FUNCTION_BLOCK MotorControla
VAR_INPUT
	Premik: BOOL;
	Smer: BOOL;
	Select: BOOL;
	KS: BOOL;
	Step: BOOL;
	Limes: WORD;
END_VAR
VAR_OUTPUT
	OutPremik: BOOL;
	OutSmer: BOOL;
	Interlock: BOOL;
	Stop: BOOL;
	Position: WORD;
END_VAR
VAR
	R_TRIG_0: R_TRIG;
	Dump: TIME;
	InL: TOF;
	RS_0: RS;

	R_TRIG_1: R_TRIG;
	TON0: TON;
	TON1: TON;
	TON_0: TON;
	Counter_0: Counter;
	F_TRIG_0: F_TRIG;
	InL1: TOF;
	IntL1: BOOL;
	IntL2: BOOL;
	IntL3: BOOL;
	R_TRIG_2: R_TRIG;
END_VAR
//dODAJ COLLISION DETECTION AND AVOIDANCE
//ZRIHTAJ SMER, KI SE SLABO SPREMINJA

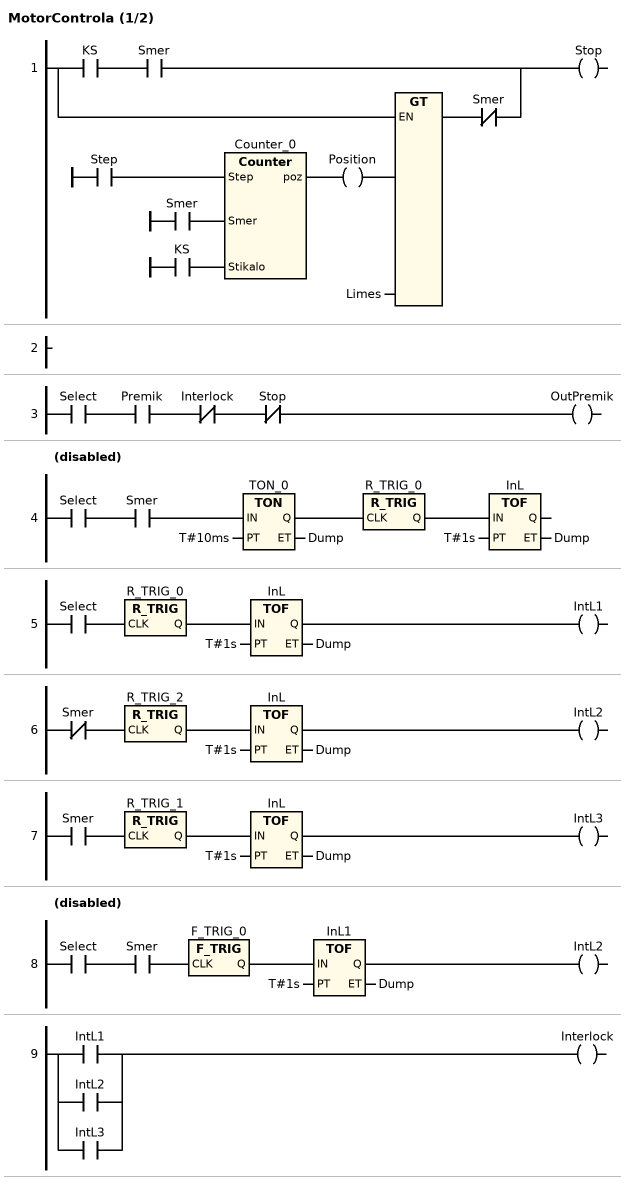
// NETWORK 1
Counter_0(Step := Step, Smer := Smer, Stikalo := KS); // Counter
Position := Counter_0.poz;
Stop := KS AND Smer OR Counter_0.poz > Limes AND NOT Smer;

// NETWORK 2

// NETWORK 3
OutPremik := Select AND Premik AND NOT Interlock AND NOT Stop;

// NETWORK 4 (disabled)
// TON_0(IN := Select AND Smer, PT := T#10ms, ET => Dump); // TON
// R_TRIG_0(CLK := TON_0.Q); // R_TRIG
// InL(IN := R_TRIG_0.Q, PT := T#1s, ET => Dump); // TOF

// NETWORK 5
R_TRIG_0(CLK := Select); // R_TRIG
InL(IN := R_TRIG_0.Q, PT := T#1s, ET => Dump); // TOF
IntL1 := InL.Q;

// NETWORK 6
R_TRIG_2(CLK := NOT Smer); // R_TRIG
InL(IN := R_TRIG_2.Q, PT := T#1s, ET => Dump); // TOF
IntL2 := InL.Q;

// NETWORK 7
R_TRIG_1(CLK := Smer); // R_TRIG
InL(IN := R_TRIG_1.Q, PT := T#1s, ET => Dump); // TOF
IntL3 := InL.Q;

// NETWORK 8 (disabled)
// F_TRIG_0(CLK := Select AND Smer); // F_TRIG
// InL1(IN := F_TRIG_0.Q, PT := T#1s, ET => Dump); // TOF
// IntL2 := InL1.Q;

// NETWORK 9
Interlock := IntL1 OR IntL2 OR IntL3;

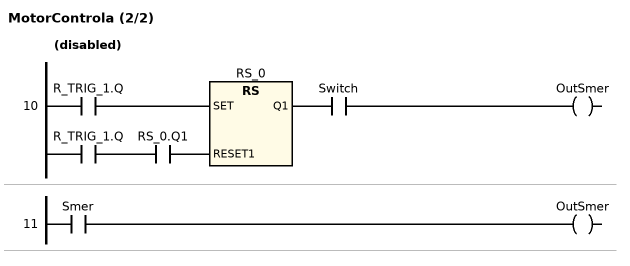
// NETWORK 10 (disabled)
// RS_0(SET := R_TRIG_1.Q, RESET1 := R_TRIG_1.Q AND RS_0.Q1); // RS
// OutSmer := RS_0.Q1 AND Switch;

// NETWORK 11
OutSmer := Smer;

END_FUNCTION_BLOCK

(* stored: Version 1.1.0.1, ProductVersion 3.1.4024.12
   POU MotorControla: Id {f931a168-8717-4e85-baf9-63ed8530a325}, SpecialFunc None *)
